TYPE TcoUrRobotics_O2TReg :
STRUCT
    {attribute addProperty Name "<#Bit registers#>"}
    Bits : ARRAY[0..31] OF BOOL;
    {attribute addProperty Name "<#Int registers#>"}
    Ints : ARRAY[0..11] OF DINT;
    {attribute addProperty Name "<#Float registers#>"}
    Floats : ARRAY[0..11] OF REAL;
END_STRUCT
END_TYPE

(* stored: Version 1.1.0.1, ProductVersion 3.1.4024.12
   DUT TcoUrRobotics_O2TReg: Id {d91d16a9-0914-0e27-0155-707ccea2a3e0} *)
